{attribute 'strict'}
{attribute 'to_string'}
TYPE E_VisuCtrlRobotImgType :
(
	ROBOT_TYPE_MITSUBISHI_6_AXIS 	:= 0,	(*  *)
	ROBOT_TYPE_MITSUBISHI_SCARA 	:= 10	(*  *)
);
END_TYPE

(* stored: Version 1.1.0.1, ProductVersion 3.1.4024.9
   DUT E_VisuCtrlRobotImgType: Id {d914421b-d3c2-42d8-816a-a1b9f675986d} *)
